Staubli VAL3: MotionCmd.pjx

--- MotionCmd.pjx ---
Parameters version=s7.7.2 stackSize=5000 millimeterUnit=true
Program file=start.pgx
Program file=stop.pgx
Data file=MotionCmd.dtx

--- MotionCmd.dtx ---
public mdesc mDesc = {leave=0, reach=0}
public num nDuration
public num nSequence
public jointRx jJointRx
